FUNCTION_BLOCK operate_IO (* Basic Function Block Type *)
  (* Standard: 61499-2 *)
  (* Version 0.0, 24/03/2016, Chen-Wei, nxtControl GmbH, Template *)
  PACKAGE Main;
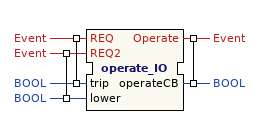
  EVENT_INPUT
    REQ WITH trip; (* Normal Execution Request *)
    REQ2 WITH lower;
  END_EVENT
  EVENT_OUTPUT
    Operate WITH operateCB; (* Execution Confirmation *)
  END_EVENT
  VAR_INPUT
    trip : BOOL;
    lower : BOOL;
  END_VAR
  VAR_OUTPUT
    operateCB : BOOL; (* Output event qualifier *)
  END_VAR
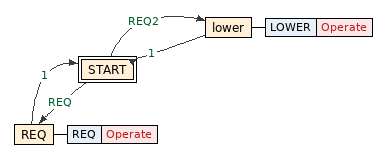
  EC_STATES
    START; (* Initial State *)
    REQ : REQ -> Operate; (* Normal execution *)
    lower : LOWER -> Operate;
  END_STATES
  EC_TRANSITIONS
    START TO REQ := REQ;
    REQ TO START := 1;
    START TO lower := REQ2;
    lower TO START := 1;
  END_TRANSITIONS
  ALGORITHM REQ IN ST: (* Normally executed algorithm *)
REQ := 0;
operateCB := trip;

;
  END_ALGORITHM
  ALGORITHM LOWER IN ST:
REQ2 := 0;

operateCB := lower;

;
  END_ALGORITHM
END_FUNCTION_BLOCK
